TYPE ST_BigBagChangeHandlerStatus :
STRUCT
    bDone               : BOOL;        // zakończona obsługa zmiany worka
    sDiag               : T_MaxString; // diagnostyka bloku
END_STRUCT
END_TYPE

(* stored: Version 1.1.0.1, ProductVersion 3.1.4024.16
   DUT ST_BigBagChangeHandlerStatus: Id {45fe3974-18f0-4864-8b5b-e453e047f122} *)
